PROGRAM MAIN
VAR
	axis1 					: AXIS_REF;
	axis2 					: AXIS_REF;
	axis3 					: AXIS_REF;
	axis4 					: AXIS_REF;
	axis5 					: AXIS_REF;
	fbPower1 				: MC_Power;
	fbPower2 				: MC_Power;
	fbPower3				: MC_Power;
	fbPower4 				: MC_Power;
	fbPower5 				: MC_Power;
	
	aEnable					: BOOL;
	fb_GearInMultiMaster	: MC_GearInMultiMaster;
	gEbable					: BOOL;
	fbMove 					: MC_MoveAbsolute;
	fbMove2 					: MC_MoveAbsolute;
	fbMove3 					: MC_MoveAbsolute;
	fbMove4 					: MC_MoveAbsolute;
oran 							: DWORD:=2;
	mEnable: BOOL;
END_VAR

//aEnable eksenleri enable etmek için ,gEbable fb_GearInMultiMaster fonksiyon bloğunu çalıştımak için, menable eksenlere hareket verebilmek için
fbPower1(
	Axis:=axis1 , 
	Enable:=aEnable, 
	Enable_Positive:= aEnable, 
	Enable_Negative:=aEnable , 
	Override:=100 );
	
fbPower2(
	Axis:=axis2 , 
	Enable:=aEnable, 
	Enable_Positive:= aEnable, 
	Enable_Negative:=aEnable , 
	Override:=100);
	
fbPower3(
	Axis:=axis3 , 
	Enable:=aEnable, 
	Enable_Positive:= aEnable, 
	Enable_Negative:=aEnable , 
	Override:=100);
	
fbPower4(
	Axis:=axis4 , 
	Enable:=aEnable, 
	Enable_Positive:= aEnable, 
	Enable_Negative:=aEnable , 
	Override:=100);
	
fbPower5(
	Axis:=axis5 , 
	Enable:=aEnable, 
	Enable_Positive:= aEnable, 
	Enable_Negative:=aEnable , 
	Override:=100);
	
	
fb_GearInMultiMaster(
	Master1:= axis1, 
	Master2:= axis2, 
	Master3:= axis3, 
	Master4:= axis4, 
	Slave  := axis5, 
	Enable := gEbable , 
	GearRatio1:= 1, 
	GearRatio2:= 2, 
	GearRatio3:= 3, 
	GearRatio4:= 4);

fbMove(
	Axis:= axis1, 
	Execute:=mEnable , 
	Position:=10 , 
	Velocity:= 10 );
	
fbMove2(
	Axis:= axis2, 
	Execute:=mEnable , 
	Position:=10 , 
	Velocity:= 10 );

fbMove3(
	Axis:= axis3, 
	Execute:=mEnable , 
	Position:=10 , 
	Velocity:= 10  );
	
fbMove4(
	Axis:= axis4, 
	Execute:=mEnable , 
	Position:=10 , 
	Velocity:= 10 );

END_PROGRAM

(* stored: Version 1.1.0.1, ProductVersion 3.1.4024.12
   POU MAIN: Id {5c50f173-78e5-4867-8be7-27e3f4f2ec7e}, SpecialFunc None *)
